Staubli VAL3: Exam_Robot.pgx

program Exam_Robot()
  local num l_LigneCurrant
begin

  call Empilement()



end
